// TIA Portal V18 export
// export: Created 2025-12-01T12:39:35.8080678Z, ExportSetting None, DisplayName Totally Integrated Automation Portal, DisplayVersion V18 Update 5, DisplayName TIA Portal Openness, DisplayVersion V18 Update 5, DisplayName TIA Portal Teamcenter Gateway, DisplayVersion V18, DisplayName TIA Portal Version Control Interface, DisplayVersion V18, DisplayName STEP 7 Professional, DisplayVersion V18 Update 5, DisplayName STEP 7 Safety, DisplayVersion V18, DisplayName WinCC Professional, DisplayVersion V18 Update 5
VAR_GLOBAL   // PLC tag table "Flow"
END_VAR
VAR_GLOBAL CONSTANT   // user constants
   station_empty : Int := 0;   // 无料
   PartStatusOK : Int := 1;   // 工件加工OK
   PartStatusNG : Int := 2;   // 工件加工NG
   MES_CheckIn_OK : Int := 100;   // 上件完成状态
   Allow_Operation : Int := 200;   // 允许装配状态
   Clean_OK : Int := 201;   // 清洗OK
   "Press_OK(1)" : Int := 202;   // 压装OK
   Process_Complete : Int := 300;   // 加工完成OK
   MES_Upload_OK : Int := 400;   // MES上传OK状态
   MES_Upload1_NG : Int := 401;   // MES上传NG状态1
   MES_Upload2_NG : Int := 402;   // MES上传NG状态2
   MES_Upload3_NG : Int := 403;   // MES上传NG状态3
   MES_Upload4_NG : Int := 404;   // MES上传NG状态4
   MES_Upload_Complete : Int := 500;   // MES上传状态完成
   LoadComplete : Int := 201;   // 单向阀上料完成
END_VAR
